% RSLogix 500 project RESFRIADOR_OLEO_BANCADA_BAK004.RSS, saved by version 8.40.00.08 %
PROJECT "UNTITLED"    % processor: Bul.1763 MicroLogix 1100 Series B %

PROGRAM FILES
  LAD 2 "PRINCIPAL"  4 rungs
  LAD 3 "COM_BOMB"  4 rungs  % comando liga bomba de oleo %
  LAD 4 "COM_VENT"  1 rungs  % comando para ligar vent %
  LAD 5 "COM_COMP"  1 rungs  % comando para ligar compressor %

DATA FILES
  O0 OUTPUT  4 elements
  I1 INPUT  6 elements
  S2 STATUS  66 elements
  B3 BINARY  1 elements
  T4 TIMER  1 elements
  C5 COUNTER  1 elements
  R6 CONTROL  1 elements
  N7 INTEGER  1 elements
  F8 FLOAT  1 elements

LADDER 2 "PRINCIPAL"
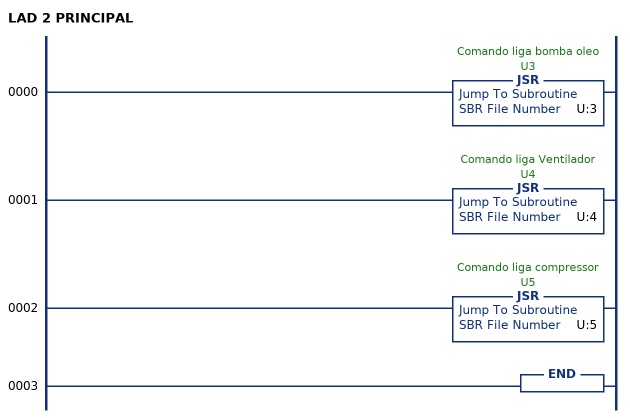
% Rung: 0 %  % edit flag set %
SOR JSR U:3 EOR
%   U:3  U3  "Comando liga bomba oleo" %
% Rung: 1 %  % edit flag set %
SOR JSR U:4 EOR
%   U:4  U4  "Comando liga Ventilador" %
% Rung: 2 %  % edit flag set %
SOR JSR U:5 EOR
%   U:5  U5  "Comando liga compressor" %
% Rung: 3 %
SOR END EOR

LADDER 3 "COM_BOMB"    % comando liga bomba de oleo %
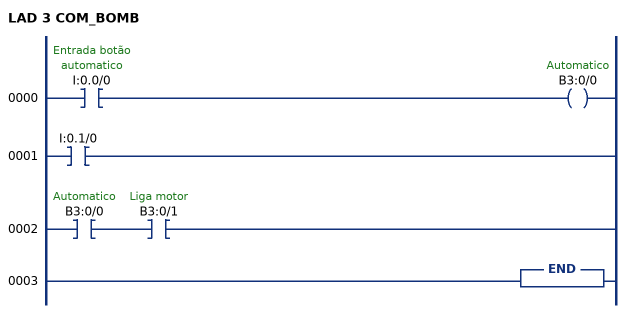
% Rung: 0 %  % edit flag set %
SOR XIC I:0.0/0 OTE B3:0/0 EOR
%   I:0.0/0  "Entrada botão automatico" %
%   B3:0/0  "Automatico" %
% Rung: 1 %  % edit flag set %
SOR XIC I:0.1/0 EOR
% Rung: 2 %  % edit flag set %
SOR XIC B3:0/0 XIC B3:0/1 EOR
%   B3:0/0  "Automatico" %
%   B3:0/1  "Liga motor" %
% Rung: 3 %
SOR END EOR
